PROGRAM MAIN
VAR
END_VAR

END_PROGRAM

(* stored: Version 1.1.0.1
   POU MAIN: Id {acbb614a-7284-4bfd-b098-a54602a5799d} *)
